(* CODESYS project timeDateTest.project

Project tree, tasks and I/O mapping:
  Device : CODESYS Control Win V3, 3S - Smart Software Solutions GmbH, order no. 305021, version 3.5.4.40
    application Application
      libraries: VisuDialogs, * (System); CmpSysExec, 1.0.0.2 (Owen); SPK_Tools, 1.0.1 (Owen); RS mode library, 1.0.0.0 (Owen); ArchiverSPK, 3.5.3.53 (Owen); CAA File, 3.5.5.0 (CAA Technical Workgroup); Time and Date, 3.5.1.0 (3S - Smart Software Solutions GmbH); Standard, * (System)
      task MainTask (cyclic, interval t#20ms, priority 1) calls PLC_PRG
      task VISU_TASK (cyclic, interval 50 ms, priority 30) calls VisuElems.Visu_Prg
      program PLC_PRG [ST]: TimeCount
      visualisation Visualization
      global variables GVL
      visualisation ManualInput
      image pool ImagePool
      visualisation Settings
      data type TableStruct
      function TimeInput [ST]
      RecipeManager
        recipe definition Receipt: PLC_PRG.arrayOfIngr[0].nameOfIngr : STRING; PLC_PRG.arrayOfIngr[0].weightOfIngr : STRING; PLC_PRG.arrayOfIngr[0].isDissolve : STRING; PLC_PRG.arrayOfIngr[0].timeOfMixing : STRING; PLC_PRG.arrayOfIngr[0].addMessage : STRING; PLC_PRG.arrayOfIngr[1].nameOfIngr : STRING; PLC_PRG.arrayOfIngr[1].weightOfIngr : STRING; PLC_PRG.arrayOfIngr[1].isDissolve : STRING; PLC_PRG.arrayOfIngr[1].timeOfMixing : STRING; PLC_PRG.arrayOfIngr[1].addMessage : STRING; PLC_PRG.arrayOfIngr[2].nameOfIngr : STRING; PLC_PRG.arrayOfIngr[2].weightOfIngr : STRING; PLC_PRG.arrayOfIngr[2].isDissolve : STRING; PLC_PRG.arrayOfIngr[2].timeOfMixing : STRING; PLC_PRG.arrayOfIngr[2].addMessage : STRING; PLC_PRG.arrayOfIngr[3].nameOfIngr : STRING; PLC_PRG.arrayOfIngr[3].weightOfIngr : STRING; PLC_PRG.arrayOfIngr[3].isDissolve : STRING; PLC_PRG.arrayOfIngr[3].timeOfMixing : STRING; PLC_PRG.arrayOfIngr[3].addMessage : STRING; PLC_PRG.arrayOfIngr[4].nameOfIngr : STRING; PLC_PRG.arrayOfIngr[4].weightOfIngr : STRING; PLC_PRG.arrayOfIngr[4].isDissolve : STRING; PLC_PRG.arrayOfIngr[4].timeOfMixing : STRING; PLC_PRG.arrayOfIngr[4].addMessage : STRING; PLC_PRG.arrayOfIngr[5].nameOfIngr : STRING; PLC_PRG.arrayOfIngr[5].weightOfIngr : STRING; PLC_PRG.arrayOfIngr[5].isDissolve : STRING; PLC_PRG.arrayOfIngr[5].timeOfMixing : STRING; PLC_PRG.arrayOfIngr[5].addMessage : STRING; PLC_PRG.arrayOfIngr[6].nameOfIngr : STRING; PLC_PRG.arrayOfIngr[6].weightOfIngr : STRING; PLC_PRG.arrayOfIngr[6].isDissolve : STRING; PLC_PRG.arrayOfIngr[6].timeOfMixing : STRING; PLC_PRG.arrayOfIngr[6].addMessage : STRING; PLC_PRG.arrayOfIngr[7].nameOfIngr : STRING; PLC_PRG.arrayOfIngr[7].weightOfIngr : STRING; PLC_PRG.arrayOfIngr[7].isDissolve : STRING; PLC_PRG.arrayOfIngr[7].timeOfMixing : STRING; PLC_PRG.arrayOfIngr[7].addMessage : STRING; PLC_PRG.arrayOfIngr[8].nameOfIngr : STRING; PLC_PRG.arrayOfIngr[8].weightOfIngr : STRING; PLC_PRG.arrayOfIngr[8].isDissolve : STRING; PLC_PRG.arrayOfIngr[8].timeOfMixing : STRING; PLC_PRG.arrayOfIngr[8].addMessage : STRING; PLC_PRG.arrayOfIngr[9].nameOfIngr : STRING; PLC_PRG.arrayOfIngr[9].weightOfIngr : STRING; PLC_PRG.arrayOfIngr[9].isDissolve : STRING; PLC_PRG.arrayOfIngr[9].timeOfMixing : STRING; PLC_PRG.arrayOfIngr[9].addMessage : STRING; PLC_PRG.arrayOfIngr[10].nameOfIngr : STRING; PLC_PRG.arrayOfIngr[10].weightOfIngr : STRING; PLC_PRG.arrayOfIngr[10].isDissolve : STRING; PLC_PRG.arrayOfIngr[10].timeOfMixing : STRING; PLC_PRG.arrayOfIngr[10].addMessage : STRING
      function two_word_to_real [ST]
      visualisation AutoWork
    Modbus_COM : Modbus COM, 3S - Smart Software Solutions GmbH, version 3.4.0.0
        settings: DataBits = 8; StopBits = 1; ComPort = 3
      Modbus_Master_COM_Port : Modbus Master, COM Port, 3S - Smart Software Solutions GmbH, version 3.5.5.0
          settings: Transmission = 'RTU'; ResponseTimeout = 300; TimeBetweenFrames = 50; Auto-restart communication = TRUE
        Modbus_Slave_COM_Port : Modbus Slave, COM Port, 3S - Smart Software Solutions GmbH, version 3.5.4.0
            settings: SlaveAddress = 16; ResponseTimeout = 300; UseExtendedFunctionCodes = TRUE; Channel 1.Function Code = 16; Channel 1.Read Offset = 0; Channel 1.Read Length = 0; Channel 1.Write Offset = 16#0032; Channel 1.Write Length = 1; Channel 1.Cycle Time = 100
            output Application.outputDiscrets : WORD  // Channel 1.Channel 1[0]
            unmapped channels: Channel 1
    Modbus_COM_1 : Modbus COM, 3S - Smart Software Solutions GmbH, version 3.4.0.0
        settings: DataBits = 8; StopBits = 1; ComPort = 4
      Modbus_Master_COM_Port_1 : Modbus Master, COM Port, 3S - Smart Software Solutions GmbH, version 3.5.5.0
          settings: Transmission = 'RTU'; ResponseTimeout = 300; TimeBetweenFrames = 50; Auto-restart communication = TRUE
        Modbus_Slave_COM_Port_1 : Modbus Slave, COM Port, 3S - Smart Software Solutions GmbH, version 3.5.4.0
            settings: SlaveAddress = 32; ResponseTimeout = 300; UseExtendedFunctionCodes = TRUE; Channel 1.Function Code = 3; Channel 1.Read Offset = 16#0046; Channel 1.Read Length = 2; Channel 1.Write Offset = 0; Channel 1.Write Length = 0; Channel 1.Cycle Time = 100; Channel 2.Function Code = 3; Channel 2.Read Offset = 16#0048; Channel 2.Read Length = 2; Channel 2.Write Offset = 0; Channel 2.Write Length = 0; Channel 2.Cycle Time = 100; Channel 3.Function Code = 3; Channel 3.Read Offset = 16#004A; Channel 3.Read Length = 2; Channel 3.Write Offset = 0; Channel 3.Write Length = 0; Channel 3.Cycle Time = 100; Channel 4.Function Code = 3; Channel 4.Read Offset = 16#004C; Channel 4.Read Length = 2; Channel 4.Write Offset = 0; Channel 4.Write Length = 0; Channel 4.Cycle Time = 100
            input  Application.arr1[0] : WORD  // Channel 1.Channel 1
            input  Application.arr1[1] : WORD  // Channel 1.Channel 1
            input  Application.arr2[0] : WORD  // Channel 2.Channel 2
            input  Application.arr2[1] : WORD  // Channel 2.Channel 2
            input  Application.arr3[0] : WORD  // Channel 3.Channel 3
            input  Application.arr3[1] : WORD  // Channel 3.Channel 3
            input  Application.arr4[0] : WORD  // Channel 4.Channel 4
            input  Application.arr4[1] : WORD  // Channel 4.Channel 4
            unmapped channels: Channel 1, Channel 2, Channel 3, Channel 4
  text list GlobalTextList
  GlobalImagePool
  image pool ImagePool
  5ce3da45-db07-42e7-a21c-a00fff4ed8f6|C:\Users\Валентин\Desktop\home.png
  5ce3da45-db07-42e7-a21c-a00fff4ed8f6|D:\Pictures\tanzania.jpg
  5ce3da45-db07-42e7-a21c-a00fff4ed8f6|D:\Pictures\tanzania800x480.jpg
  5ce3da45-db07-42e7-a21c-a00fff4ed8f6|D:\Pictures\BeachHouse800x480.jpg
  5ce3da45-db07-42e7-a21c-a00fff4ed8f6|D:\Projects\OWEN\JAVA\GIT\settings.png
  5ce3da45-db07-42e7-a21c-a00fff4ed8f6|D:\Projects\OWEN\PIC\motherboard.png
  5ce3da45-db07-42e7-a21c-a00fff4ed8f6|D:\Projects\OWEN\PIC\home.png
  5ce3da45-db07-42e7-a21c-a00fff4ed8f6|D:\Projects\OWEN\PIC\settings.jpg
  5ce3da45-db07-42e7-a21c-a00fff4ed8f6|D:\Projects\OWEN\PIC\reset.jpg
  5ce3da45-db07-42e7-a21c-a00fff4ed8f6|D:\Projects\OWEN\PIC\reset.png
  5ce3da45-db07-42e7-a21c-a00fff4ed8f6|D:\Projects\OWEN\PIC\resetButton.png
  5ce3da45-db07-42e7-a21c-a00fff4ed8f6|D:\Projects\OWEN\PIC\start.png
  5ce3da45-db07-42e7-a21c-a00fff4ed8f6|D:\Projects\OWEN\PIC\remove.png
  5ce3da45-db07-42e7-a21c-a00fff4ed8f6|D:\Projects\OWEN\PIC\ok.png
  5ce3da45-db07-42e7-a21c-a00fff4ed8f6|D:\Projects\OWEN\PIC\cancel.png
  function block Time_Struct [ST]
  5ce3da45-db07-42e7-a21c-a00fff4ed8f6|D:\Projects\OWEN\PIC\add.png
  5ce3da45-db07-42e7-a21c-a00fff4ed8f6|D:\Projects\OWEN\PIC\back.png
  5ce3da45-db07-42e7-a21c-a00fff4ed8f6|D:\Projects\OWEN\PIC\next.png
  5ce3da45-db07-42e7-a21c-a00fff4ed8f6|D:\Projects\OWEN\PIC\Drives-Downloads-icon.png
  5ce3da45-db07-42e7-a21c-a00fff4ed8f6|D:\Projects\OWEN\PIC\Actions-application-exit-icon.png
  5ce3da45-db07-42e7-a21c-a00fff4ed8f6|D:\Projects\OWEN\PIC\App-desktop-enhancements-icon.png
  5ce3da45-db07-42e7-a21c-a00fff4ed8f6|D:\Projects\OWEN\PIC\chemistryS.png
  5ce3da45-db07-42e7-a21c-a00fff4ed8f6|D:\Projects\OWEN\PIC\chemistry.png
  5ce3da45-db07-42e7-a21c-a00fff4ed8f6|D:\Projects\OWEN\PIC\Iconshock-Real-Vista-Education-Laboratory.png
*)

// Device/Application/TableStruct
TYPE TableStruct :
STRUCT
	nameOfIngr:STRING;
	weightOfIngr:STRING;
	isDissolve:STRING;
	timeOfMixing:STRING;
	addMessage:STRING;
	
END_STRUCT
END_TYPE

// Device/Application/GVL
VAR_GLOBAL
	outputDiscrets: INT;
	arr1:ARRAY[0..1]OF WORD;		
	arr2:ARRAY[0..1]OF WORD;
	arr3:ARRAY[0..1]OF WORD;
	arr4:ARRAY[0..1]OF WORD;
	
	
END_VAR

// Device/Application/PLC_PRG
PROGRAM PLC_PRG
VAR
	down: STRING;
	crntTimer:TIME;
	strTimer:STRING;
	currentTime:TIME;
	testWordVar:WORD := 60;
	
	prgAmount:INT:=100;
	resipeExt: STRING :='Receipt';
	RecManager 		: RecipeManCommands;
	ListOfPrgNames: ARRAY[0..100] OF STRING;
	idxOfPrgList:INT;
	ptToListPrg: POINTER TO ARRAY [0..100] OF STRING := ADR(ListOfPrgNames);
	
//----------------------------------------------------------------\\	
	data0:real;
	data1:WORD;
	init:BOOL:=TRUE;
	download:BOOL;
	save:BOOL;
	ingrArrayLength: INT := 10;
	arrayOfIngr: ARRAY[0..10] OF TableStruct;
	x: INT := 0;
	edge: INT := 1000;
	light: BOOL;
	swich: BOOL;	
	lamp1: BOOL := outputDiscrets.0;
	increment: INT := 1;	
	manualButtonStart: BOOL;
	testButton: BOOL;
	cleanCounter:INT;
END_VAR
VAR RETAIN	
	writeToTable:BOOL;
	idxOfLine:INT := 0;
	currentPrgName: STRING;
	fileName: STRING;
	currentIngredientName: STRING;
	inputTime:DWORD;	
	currentTimeMixing: TIME;
	maximumWeight: INT := 1000;
	currentWeight: INT;
	currentPoint : INT;
	manualMode: BOOL;
	dissolve: BOOL;
	message: STRING;
END_VAR

IF init = TRUE THEN	
	crntTimer:=TimeInput(testWordVar);
	RecManager.ReloadRecipes(resipeExt);
	RecManager.GetRecipeNames(resipeExt, ptToListPrg, 100,0);	
	init:=FALSE;
END_IF

TimeCount();

data0:=two_word_to_real(ADR(arr1));
data1:=arr1[1];
IF lamp1 = TRUE THEN
	outputDiscrets.0:=TRUE;
	ELSE
	outputDiscrets.0:=FALSE;
END_IF
IF writeTotable = TRUE THEN
	arrayOfIngr[idxOfLine].nameOfIngr:=currentIngredientName;
	arrayOfIngr[idxOfLine].weightOfIngr:=INT_TO_STRING(currentWeight);
	arrayOfIngr[idxOfLine].isDissolve:=BOOL_TO_STRING(dissolve);
	currentTimeMixing:=TimeInput(inputTime);
	arrayOfIngr[idxOfLine].timeOfMixing:=TIME_TO_STRING(currentTimeMixing);
	arrayOfIngr[idxOfLine].addMessage:=message;
	idxOfLine := idxOfLine + 1;		
	writeTotable:=FALSE;
	IF idxOfLine > ingrArrayLength THEN
		idxOfLine := 0;
	END_IF
END_IF

IF swich = TRUE THEN
x := x + increment;
light := TRUE;
 IF x >= currentWeight + currentPoint THEN 
	 currentPoint:= currentPoint+currentWeight;
	 increment:=0;
 outputDiscrets.0:=TRUE; 
 swich:= FALSE; 
 END_IF	 		
END_IF

IF manualMode = TRUE THEN
	swich:=TRUE;
END_IF

ACTION TimeCount:
IF TIME_TO_REAL(crntTimer) > 0 THEN
  crntTimer := REAL_TO_TIME ( TIME_TO_REAL(crntTimer) - 20);
END_IF
strTimer:=TIME_TO_STRING(crntTimer);
END_ACTION

END_PROGRAM

// Device/Application/TimeInput
FUNCTION TimeInput : TIME
VAR_INPUT
	timeSet:DWORD;	
END_VAR
VAR		
END_VAR

TimeInput:=DWORD_TO_TIME(timeSet * 1000);

END_FUNCTION

// Device/Application/two_word_to_real
FUNCTION two_word_to_real : REAL
VAR_INPUT
	in_data: POINTER TO ARRAY[0..1]OF WORD;
END_VAR
VAR
	p1:POINTER TO BYTE;
	p2:POINTER TO BYTE;
END_VAR

p1:=ADR(two_word_to_real);
p2:=ADR(in_data^[1]);

p1^:=p2^;
p1:=p1+1;
p2:=p2+1;
p1^:=p2^;
p1:=p1+1;
p2:=ADR(in_data^[0]);
p1^:=p2^;
p1:=p1+1;
p2:=p2+1;
p1^:=p2^;

END_FUNCTION

// Time_Struct
FUNCTION_BLOCK Time_Struct
VAR_INPUT
	Type_Time:TIME;
END_VAR
VAR_OUTPUT
	Day:DWORD;
	Hour:DWORD;
	Minute:DWORD;
	Second:DWORD;
	Millisecond:DWORD;  
END_VAR
VAR
		Time_DWORD:DWORD;
		Day_Ost:DWORD;
		Hour_Ost:DWORD;
		Minute_Ost:DWORD;
		Second_Ost:DWORD;
		Millisecond_Ost:DWORD; 
END_VAR


Time_DWORD := TIME_TO_DWORD(Type_Time);

Millisecond := Second_Ost;

Second := Minute_Ost/ 1000;
Second_Ost := Minute_Ost MOD 1000;

Minute := Hour_Ost/60000;
Minute_Ost := Hour_Ost MOD 60000;

Hour := Day_Ost/3600000;
Hour_Ost := Day_Ost MOD 3600000;

Day := Time_DWORD/86400000;
Day_Ost := Time_DWORD MOD 86400000;

END_FUNCTION_BLOCK

// Device/Application/Visualization
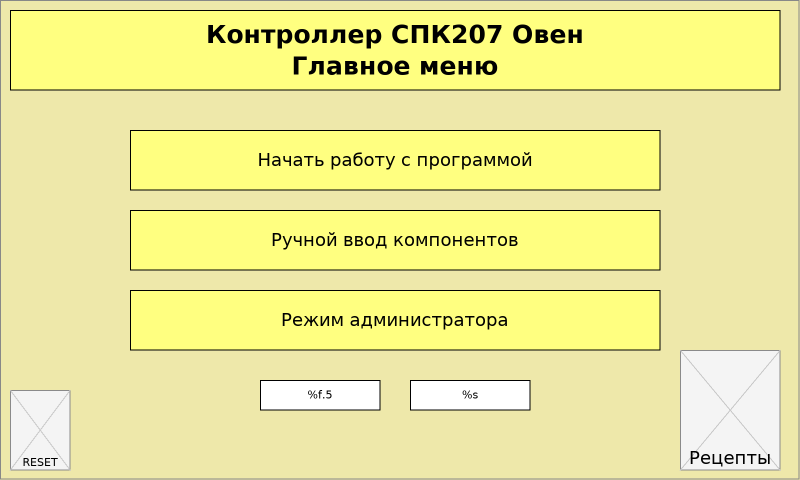
VISUALIZATION Visualization  // 800x480
    Image (10,390 60x80), "RESET", image: ImagePool.start
        OnMouseClick: execute {
            //SysExecute('/sbin/reboot');
        }
    Image (680,350 100x120), "Рецепты", image: ImagePool.Iconshock-Real-Vista-Education-Laboratory
        OnMouseClick:  Assign=Settings, Type=Assignment
    RoundedRectangle (10,10 770x80), "Контроллер СПК207 Овен Главное меню"
    RoundedRectangle (130,130 530x60), "Начать работу с программой"
        OnMouseClick:  Assign=AutoWork, Type=Assignment
        OnMouseClick:  ToggleVariable=PLC_PRG.init
    RoundedRectangle (130,210 530x60), "Ручной ввод компонентов"
        OnMouseClick:  Assign=ManualInput, Type=Assignment
        OnMouseClick: execute { PLC_PRG.manualMode:=true; }
    RoundedRectangle (130,290 530x60), "Режим администратора"
        OnMouseClick:  Type=Login
    RoundedRectangle (260,380 120x30), "%f.5", text variable: PLC_PRG.data0
    RoundedRectangle (410,380 120x30), "%s", text variable: PLC_PRG.strTimer
END_VISUALIZATION

// Device/Application/ManualInput
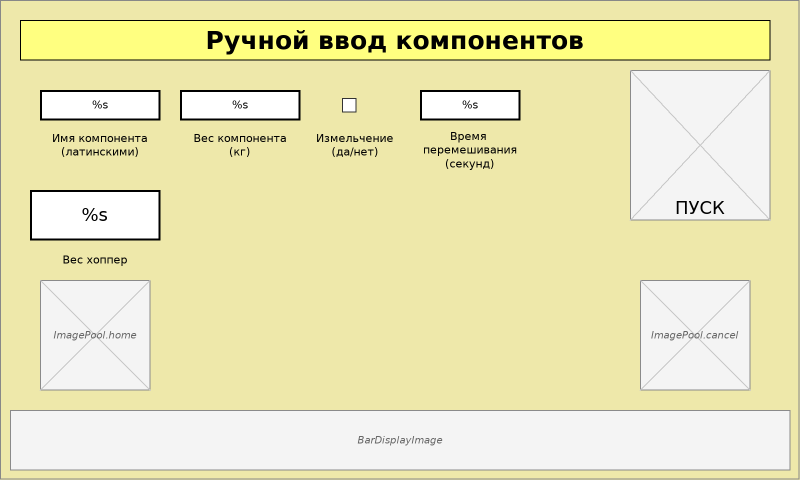
VISUALIZATION ManualInput  // 800x480
    RoundedRectangle (20,20 750x40), "Ручной ввод компонентов"
    RoundedRectangle (180,90 120x30), "%s", text variable: PLC_PRG.currentWeight
        OnMouseClick: execute { PLC_PRG.edge:=PLC_PRG.maximumWeight -PLC_PRG.x; }
        OnMouseClick: write PLC_PRG.currentWeight via VisuDialogs.Numpad, min 10, max PLC_PRG.edge
    RoundedRectangle (180,130 120x30), "Вес компонента (кг)"
    RoundedRectangle (300,130 110x30), "Измельчение (да/нет)"
    RoundedRectangle (420,90 100x30), "%s", text variable: PLC_PRG.currentTime, colour toggle: PLC_PRG.testButton
        OnMouseClick: write PLC_PRG.inputTime via VisuDialogs.Numpad, min 0
    RoundedRectangle (400,130 140x40), "Время перемешивания (секунд)"
    Image (630,70 140x150), "ПУСК", image: ImagePool.ok
        OnMouseClick:  ToggleVariable=PLC_PRG.swich
        OnMouseClick: execute {
            IF PLC_PRG.currentWeight > 0
            THEN PLC_PRG.increment:=1;
            END_IF
            PLC_PRG.currentTimeMixing:=
            TimeInput(PLC_PRG.inputTime);
        }
    BarDisplayImage (10,410 780x60), value: PLC_PRG.x, style: BarDisplayImage-Gray, scale format: %.0f, scale 0..1000
    RoundedRectangle (30,190 130x50), "%s", text variable: PLC_PRG.x
        OnMouseClick: execute { PLC_PRG.edge:=PLC_PRG.maximumWeight -PLC_PRG.x; }
        OnMouseClick: write PLC_PRG.currentWeight via VisuDialogs.Numpad, min 10, max PLC_PRG.edge
    Image (40,280 110x110), image: ImagePool.home
        OnMouseClick:  Assign=Visualization, Type=Assignment
        OnMouseClick: execute { PLC_PRG.manualMode:=false; }
    Image (640,280 110x110), image: ImagePool.cancel
        OnMouseClick: execute {
            PLC_PRG.x:=0;
            PLC_PRG.currentWeight:=0;
            PLC_PRG.currentPoint:=0;
        }
    RoundedRectangle (40,90 120x30), "%s", text variable: PLC_PRG.currentIngredientName
        OnMouseClick: write the text variable via VisuDialogs.Keypad, min 1, max 30
    RoundedRectangle (40,130 120x30), "Имя компонента (латинскими)"
    RoundedRectangle (30,250 130x20), "Вес хоппер"
    Checkbox (340,90 30x30), variable: PLC_PRG.dissolve
END_VISUALIZATION

// Device/Application/Settings
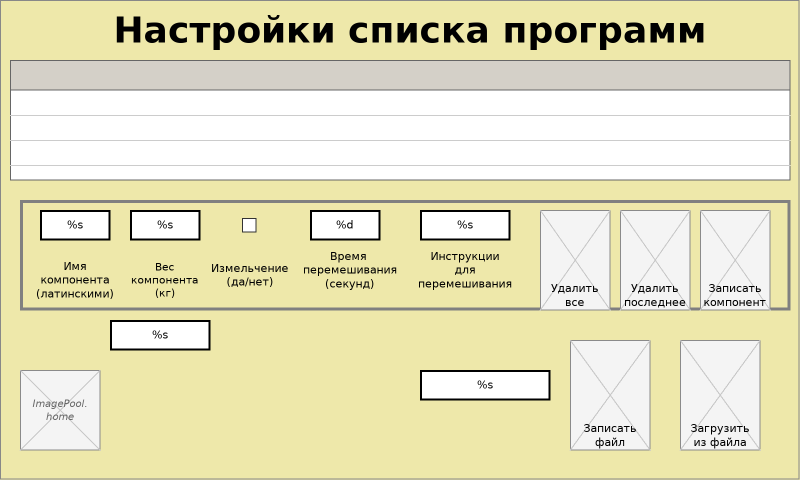
VISUALIZATION Settings  // 800x480
    Rectangle (70,10 680x40), "Настройки списка программ"
    Image (20,370 80x80), image: ImagePool.home
        OnMouseClick:  Assign=Visualization, Type=Assignment
    Table (10,60 780x120), data array: PLC_PRG.arrayOfIngr
        p1128707560: PLC_PRG.ingrArrayLength
        p3854506369: PLC_PRG.arrayOfIngr[INDEX].nameOfIngr
        p1892666644: PLC_PRG.arrayOfIngr[INDEX].weightOfIngr
        p338671338: PLC_PRG.arrayOfIngr[INDEX].isDissolve
        p2170511999: PLC_PRG.arrayOfIngr[INDEX].timeOfMixing
        p3723444502: PLC_PRG.arrayOfIngr[INDEX].addMessage
        p2232123230: Name of the ingredient
        p1755163831: is dissolve
        p1137915858: PLC_PRG.idxOfLine
    Rectangle (20,200 770x110)
    RoundedRectangle (130,210 70x30), "%s", text variable: PLC_PRG.currentWeight
        OnMouseClick: execute { PLC_PRG.edge:=PLC_PRG.maximumWeight -PLC_PRG.x; }
        OnMouseClick: write PLC_PRG.currentWeight via VisuDialogs.Numpad, min 10, max PLC_PRG.edge
    RoundedRectangle (130,250 70x60), "Вес компонента (кг)"
    RoundedRectangle (210,250 80x50), "Измельчение (да/нет)"
    RoundedRectangle (310,210 70x30), "%d", text variable: PLC_PRG.inputTime, colour toggle: PLC_PRG.testButton
        OnMouseClick: write the text variable via VisuDialogs.Numpad, min 0
    RoundedRectangle (300,250 100x40), "Время перемешивания (секунд)"
    RoundedRectangle (40,210 70x30), "%s", text variable: PLC_PRG.currentIngredientName
        OnMouseClick: write the text variable via VisuDialogs.Keypad, min 1, max 30
    RoundedRectangle (30,250 90x60), "Имя компонента (латинскими)"
    Checkbox (240,210 30x30), variable: PLC_PRG.dissolve
    RoundedRectangle (420,210 90x30), "%s", text variable: PLC_PRG.message
        OnMouseClick: write the text variable via VisuDialogs.Keypad, min 1, max 30
    RoundedRectangle (410,250 110x40), "Инструкции для перемешивания"
    Image (570,340 80x110), "Записать файл", image: ImagePool.Drives-Downloads-icon
        OnMouseClick:  ExecuteCommand=ExecuteCommand=[Command=CreateRecipe, Value='Receipt', Value2=PLC_PRG.currentPrgName, Command=SaveRecipeAs, Value='Receipt', Value2=PLC_PRG.currentPrgName]
    Image (680,340 80x110), "Загрузить из файла", image: ImagePool.App-desktop-enhancements-icon
        OnMouseClick:  ExecuteCommand=ExecuteCommand=[Command=LoadRecipeFrom, Value='Receipt']
    RoundedRectangle (110,320 100x30), "%s", text variable: PLC_PRG.currentPrgName
        OnMouseClick: write the text variable via VisuDialogs.Keypad, min 1, max 30
    Image (540,210 70x100), "Удалить все", image: ImagePool.cancel
        OnMouseClick: execute {
            FOR PLC_PRG.cleanCounter:=0 TO PLC_PRG.ingrArrayLength DO
            	PLC_PRG.arrayOfIngr[PLC_PRG.cleanCounter].nameOfIngr:='';
            	PLC_PRG.arrayOfIngr[PLC_PRG.cleanCounter].weightOfIngr:='';
            	PLC_PRG.arrayOfIngr[PLC_PRG.cleanCounter].isDissolve:='';
            	PLC_PRG.arrayOfIngr[PLC_PRG.cleanCounter].timeOfMixing:='';
            	PLC_PRG.arrayOfIngr[PLC_PRG.cleanCounter].addMessage:='';
            END_FOR
             PLC_PRG.cleanCounter:=0;
             PLC_PRG.idxOfLine:=0;
        }
    Image (620,210 70x100), "Удалить последнее", image: ImagePool.remove
        OnMouseClick: execute {
            IF PLC_PRG.idxOfLine > 0 THEN
             PLC_PRG.idxOfLine:=PLC_PRG.idxOfLine - 1;
             END_IF
            	PLC_PRG.arrayOfIngr[PLC_PRG.idxOfLine].nameOfIngr:='';
            	PLC_PRG.arrayOfIngr[PLC_PRG.idxOfLine].weightOfIngr:='';
            	PLC_PRG.arrayOfIngr[PLC_PRG.idxOfLine].isDissolve:='';
            	PLC_PRG.arrayOfIngr[PLC_PRG.idxOfLine].timeOfMixing:='';
            	PLC_PRG.arrayOfIngr[PLC_PRG.idxOfLine].addMessage:='';
        }
    Image (700,210 70x100), "Записать компонент", image: ImagePool.add
        OnMouseClick:  ToggleVariable=PLC_PRG.writeToTable
    RoundedRectangle (420,370 130x30), "%s", text variable: PLC_PRG.currentPrgName
        OnMouseClick: write the text variable via VisuDialogs.Keypad, min 1, max 30
END_VISUALIZATION

// Device/Application/AutoWork
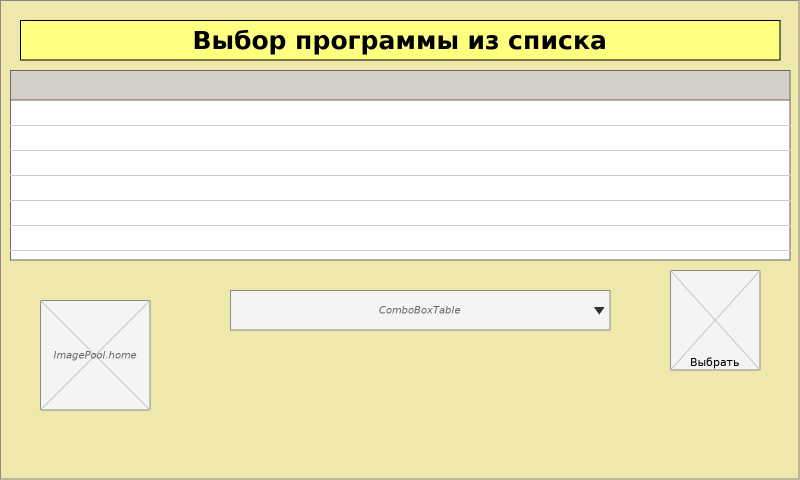
VISUALIZATION AutoWork  // 800x480
    RoundedRectangle (20,20 760x40), "Выбор программы из списка"
    ComboBoxTable (230,290 380x40), variable: PLC_PRG.idxOfPrgList, data array: PLC_PRG.ListOfPrgNames
        p3854506369: PLC_PRG.ListOfPrgNames[INDEX]
    Image (40,300 110x110), image: ImagePool.home
        OnMouseClick:  Assign=Visualization, Type=Assignment
        OnMouseClick: execute { PLC_PRG.manualMode:=false; }
    Image (670,270 90x100), "Выбрать", image: ImagePool.ok
        OnMouseClick:  ExecuteCommand=ExecuteCommand=[Command=WriteRecipe, Value='Receipt', Value2=PLC_PRG.ListOfPrgNames[PLC_PRG.idxOfPrgList]]
    Table (10,70 780x190), data array: PLC_PRG.arrayOfIngr
        p1128707560: PLC_PRG.ingrArrayLength
        p3854506369: PLC_PRG.arrayOfIngr[INDEX].nameOfIngr
        p1892666644: PLC_PRG.arrayOfIngr[INDEX].weightOfIngr
        p338671338: PLC_PRG.arrayOfIngr[INDEX].isDissolve
        p2170511999: PLC_PRG.arrayOfIngr[INDEX].timeOfMixing
        p3723444502: PLC_PRG.arrayOfIngr[INDEX].addMessage
        p2232123230: Name of the ingredient
        p1755163831: is dissolve
END_VISUALIZATION
